{attribute 'linkalways'} 
{attribute 'no_explicit_call' := 'This FB is a CLASS and must be accessed using methods or properties'}
{attribute 'enable_dynamic_creation'}
FUNCTION_BLOCK FINAL Node_LREAL_TO_UDINT EXTENDS Node
VAR
	in : _LREAL(0.0);
	out : _UDINT(0);
	success : _BOOL(FALSE);
END_VAR

METHOD PUBLIC  Clone : I_Node
VAR
	pNode : POINTER TO Node_LREAL_TO_UDINT;
END_VAR
pNode := __NEW(Node_LREAL_TO_UDINT);
Clone := pNode^;
END_METHOD

METHOD FB_init : BOOL
VAR_INPUT
	bInitRetains : BOOL; // if TRUE, the retain variables are initialized (warm start / cold start)
	bInCopyCode : BOOL;  // if TRUE, the instance afterwards gets moved into the copy code (online change)
END_VAR
AddParameter('in', in);
AddOutput('out', out);
AddOutput('success', success);

this^.Metadatum.AddBoolAsMetadata('deprecated', true);
END_METHOD

METHOD PROTECTED OnExecute
VAR
END_VAR
success.Value := TryConvert_LREAL_TO_UDINT(in.Value, out.Value);
END_METHOD

END_FUNCTION_BLOCK

(* stored: Version 1.1.0.1, ProductVersion 3.1.4026.18
   POU Node_LREAL_TO_UDINT: Id {25880341-042f-0a26-347e-c6ad0d3262d2}, SpecialFunc None
   Folder Constructor: Id {654f4667-3e73-0f25-06a8-906a25a6cd21}
   Method Clone: Id {1dea47d1-9ff4-05d9-324f-a71da0bb7e39}
   Method FB_init: Id {5327b1d5-a9cf-0dfd-23db-3fd1426c4f9b}
   Method OnExecute: Id {2016caf2-dc16-0e7c-1f04-28f9ca79b901} *)
